{attribute 'qualified_only'}
VAR_GLOBAL
	P1: BOOL; 	// "Pumpe Ein"
	P2: BOOL;   // "Störung"
	Q1: BOOL;   // Motor Pumpe
END_VAR

(* stored: Version 1.1.0.1, ProductVersion 3.1.4024.4
   GVL SimDA: Id {efa3d63a-96e1-4204-b1e7-9f3703bd4f03} *)
